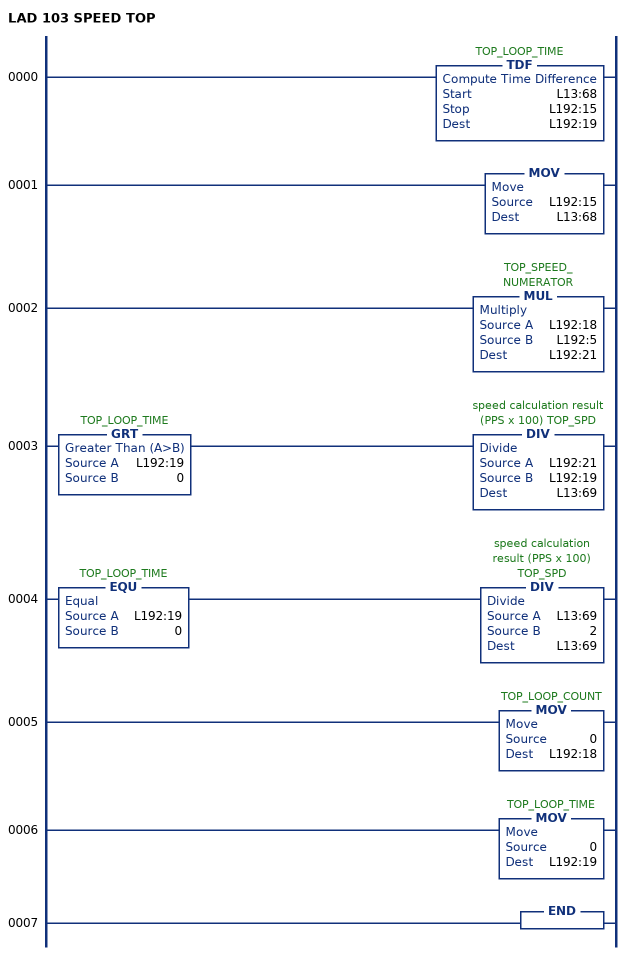
% Rung: 0 %
SOR TDF L13:68 L192:15 L192:19 EOR
%   L192:15  TOP_THIS_TIME  "rtc top belt movement event time" %
%   L192:19  TOP_LOOP_TIME %
% Rung: 1 %
SOR MOV L192:15 L13:68 EOR
%   L192:15  TOP_THIS_TIME  "rtc top belt movement event time" %
% Rung: 2 %
SOR MUL L192:18 L192:5 L192:21 EOR
%   L192:18  TOP_LOOP_COUNT %
%   L192:5  TKS_PER_SECOND %
%   L192:21  TOP_SPEED_NUMERATOR %
% Rung: 3 %
SOR GRT L192:19 0 DIV L192:21 L192:19 L13:69 EOR
%   L192:19  TOP_LOOP_TIME %
%   L192:21  TOP_SPEED_NUMERATOR %
%   L13:69  TOP_SPD  "speed calculation result (PPS x 100)" %
% Rung: 4 %
SOR EQU L192:19 0 DIV L13:69 2 L13:69 EOR
%   L192:19  TOP_LOOP_TIME %
%   L13:69  TOP_SPD  "speed calculation result (PPS x 100)" %
% Rung: 5 %
SOR MOV 0 L192:18 EOR
%   L192:18  TOP_LOOP_COUNT %
% Rung: 6 %
SOR MOV 0 L192:19 EOR
%   L192:19  TOP_LOOP_TIME %
% Rung: 7 %
SOR END EOR

LADDER 105 "P TOP"    % high speed %
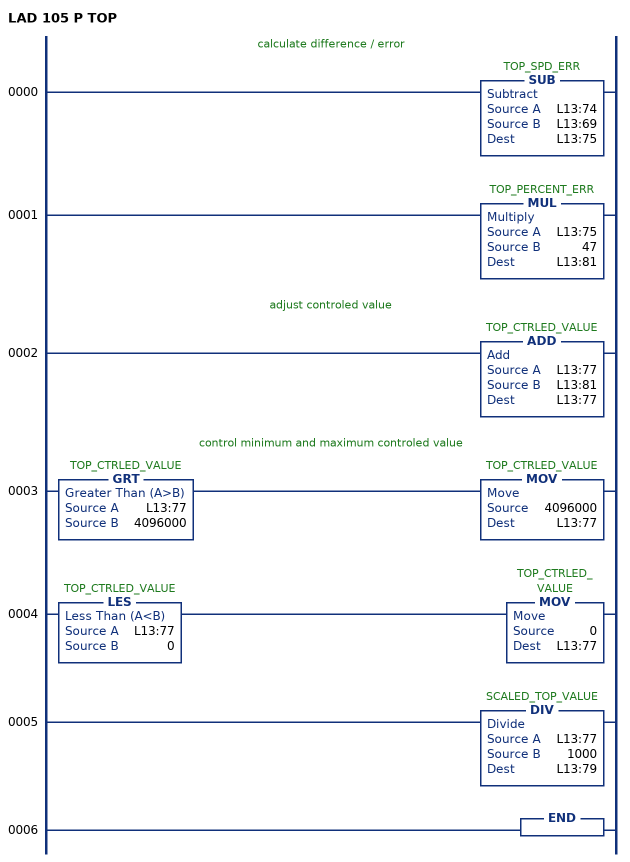
% Rung: 0 %
% calculate difference / error %
SOR SUB L13:74 L13:69 L13:75 EOR
%   L13:74  TOP_SPD_SETPOINT %
%   L13:69  TOP_SPD  "speed calculation result (PPS x 100)" %
%   L13:75  TOP_SPD_ERR %
% Rung: 1 %
SOR MUL L13:75 47 L13:81 EOR
%   L13:75  TOP_SPD_ERR %
%   L13:81  TOP_PERCENT_ERR %
% Rung: 2 %
% adjust controled value %
SOR ADD L13:77 L13:81 L13:77 EOR
%   L13:77  TOP_CTRLED_VALUE %
%   L13:81  TOP_PERCENT_ERR %
% Rung: 3 %
% control minimum and maximum controled value %
SOR GRT L13:77 4096000 MOV 4096000 L13:77 EOR
%   L13:77  TOP_CTRLED_VALUE %
% Rung: 4 %
SOR LES L13:77 0 MOV 0 L13:77 EOR
%   L13:77  TOP_CTRLED_VALUE %
% Rung: 5 %
SOR DIV L13:77 1000 L13:79 EOR
%   L13:77  TOP_CTRLED_VALUE %
%   L13:79  SCALED_TOP_VALUE %
% Rung: 6 %
SOR END EOR

LADDER 111 "SHIFT TOP"
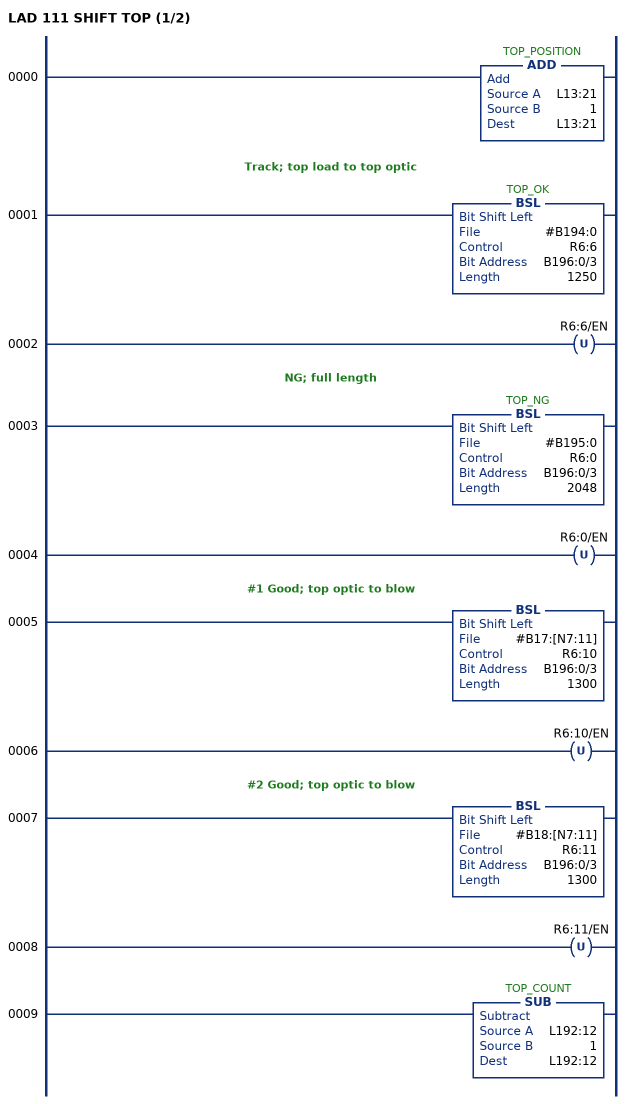
% Rung: 0 %
SOR ADD L13:21 1 L13:21 EOR
%   L13:21  TOP_POSITION %
% Rung: 1 %
% TITLE: Track; top load to top optic %
SOR BSL #B194:0 R6:6 B196:0/3 1250 EOR
%   B194:0  TOP_OK %
%   B196:0/3  OFF %
% Rung: 2 %
SOR OTU R6:6/EN EOR
% Rung: 3 %
% TITLE: NG; full length %
SOR BSL #B195:0 R6:0 B196:0/3 2048 EOR
%   B195:0  TOP_NG %
%   B196:0/3  OFF %
% Rung: 4 %
SOR OTU R6:0/EN EOR
% Rung: 5 %
% TITLE: #1 Good; top optic to blow %
SOR BSL #B17:[N7:11] R6:10 B196:0/3 1300 EOR
%   B196:0/3  OFF %
% Rung: 6 %
SOR OTU R6:10/EN EOR
% Rung: 7 %
% TITLE: #2 Good; top optic to blow %
SOR BSL #B18:[N7:11] R6:11 B196:0/3 1300 EOR
%   B196:0/3  OFF %
% Rung: 8 %
SOR OTU R6:11/EN EOR
% Rung: 9 %
SOR SUB L192:12 1 L192:12 EOR
%   L192:12  TOP_COUNT %

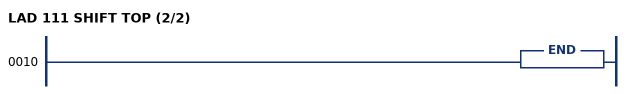
% Rung: 10 %
SOR END EOR

LADDER 131 "READXFER"
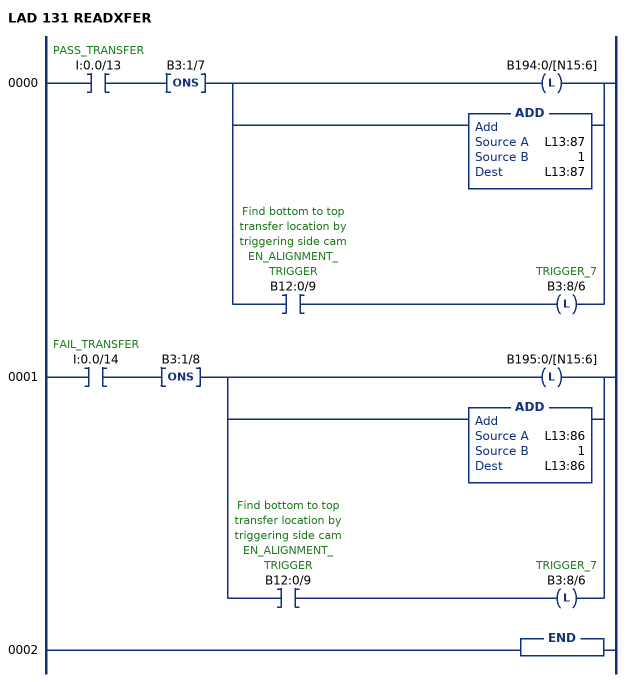
% Rung: 0 %
SOR XIC I:0.0/13 ONS B3:1/7 BST OTL B194:0/[N15:6] NXB ADD L13:87 1 L13:87 NXB XIC B12:0/9 OTL B3:8/6 BND EOR
%   I:0.0/13  PASS_TRANSFER %
%   B194:0  TOP_OK %
%   N15:6  XFER_IN_LOC %
%   B12:0/9  EN_ALIGNMENT_TRIGGER  "Find bottom to top transfer location by triggering side cam" %
%   B3:8/6  TRIGGER_7 %
% Rung: 1 %
SOR XIC I:0.0/14 ONS B3:1/8 BST OTL B195:0/[N15:6] NXB ADD L13:86 1 L13:86 NXB XIC B12:0/9 OTL B3:8/6 BND EOR
%   I:0.0/14  FAIL_TRANSFER %
%   B195:0  TOP_NG %
%   N15:6  XFER_IN_LOC %
%   B12:0/9  EN_ALIGNMENT_TRIGGER  "Find bottom to top transfer location by triggering side cam" %
%   B3:8/6  TRIGGER_7 %
% Rung: 2 %
SOR END EOR

LADDER 138 "BYPASTOPOP"
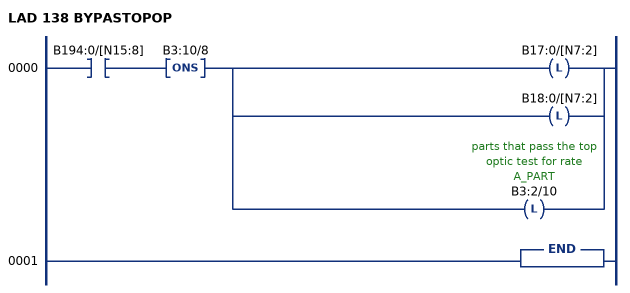
% Rung: 0 %
SOR XIC B194:0/[N15:8] ONS B3:10/8 BST OTL B17:0/[N7:2] NXB OTL B18:0/[N7:2] NXB OTL B3:2/10 BND EOR
%   B194:0  TOP_OK %
%   N15:8  TOP_OPTIC_LOC %
%   B17:0  GOOD1 %
%   N7:2  TOP_OPT_LOAD_LOC  "part load location" %
%   B18:0  GOOD2 %
%   B3:2/10  A_PART  "parts that pass the top optic test for rate" %
% Rung: 1 %
SOR END EOR

LADDER 140 "TOP_OPTIC"
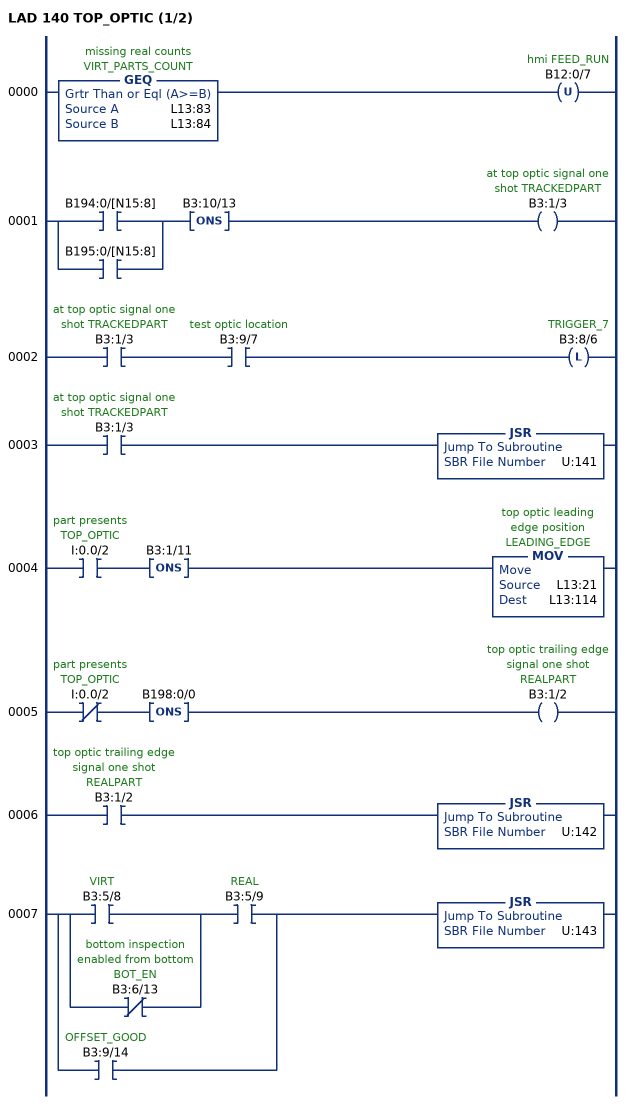
% Rung: 0 %
SOR GEQ L13:83 L13:84 OTU B12:0/7 EOR
%   L13:83  VIRT_PARTS_COUNT  "missing real counts" %
%   L13:84  FELL_PARTS_LIMIT %
%   B12:0/7  FEED_RUN  "hmi" %
% Rung: 1 %
SOR BST XIC B194:0/[N15:8] NXB XIC B195:0/[N15:8] BND ONS B3:10/13 OTE B3:1/3 EOR
%   B194:0  TOP_OK %
%   N15:8  TOP_OPTIC_LOC %
%   B195:0  TOP_NG %
%   B3:1/3  TRACKEDPART  "at top optic signal one shot" %
% Rung: 2 %
SOR XIC B3:1/3 XIC B3:9/7 OTL B3:8/6 EOR
%   B3:1/3  TRACKEDPART  "at top optic signal one shot" %
%   B3:9/7  "test optic location" %
%   B3:8/6  TRIGGER_7 %
% Rung: 3 %
SOR XIC B3:1/3 JSR U:141 EOR
%   B3:1/3  TRACKEDPART  "at top optic signal one shot" %
% Rung: 4 %
SOR XIC I:0.0/2 ONS B3:1/11 MOV L13:21 L13:114 EOR
%   I:0.0/2  TOP_OPTIC  "part presents" %
%   L13:21  TOP_POSITION %
%   L13:114  LEADING_EDGE  "top optic leading edge position" %
% Rung: 5 %
SOR XIO I:0.0/2 ONS B198:0/0 OTE B3:1/2 EOR
%   I:0.0/2  TOP_OPTIC  "part presents" %
%   B3:1/2  REALPART  "top optic trailing edge signal one shot" %
% Rung: 6 %
SOR XIC B3:1/2 JSR U:142 EOR
%   B3:1/2  REALPART  "top optic trailing edge signal one shot" %
% Rung: 7 %
SOR BST BST XIC B3:5/8 NXB XIO B3:6/13 BND XIC B3:5/9 NXB XIC B3:9/14 BND JSR U:143 EOR
%   B3:5/8  VIRT %
%   B3:6/13  BOT_EN  "bottom inspection enabled from bottom" %
%   B3:5/9  REAL %
%   B3:9/14  OFFSET_GOOD %

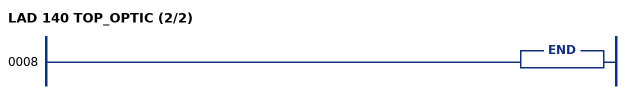
% Rung: 8 %
SOR END EOR

LADDER 141 "TOPOP_VERT"
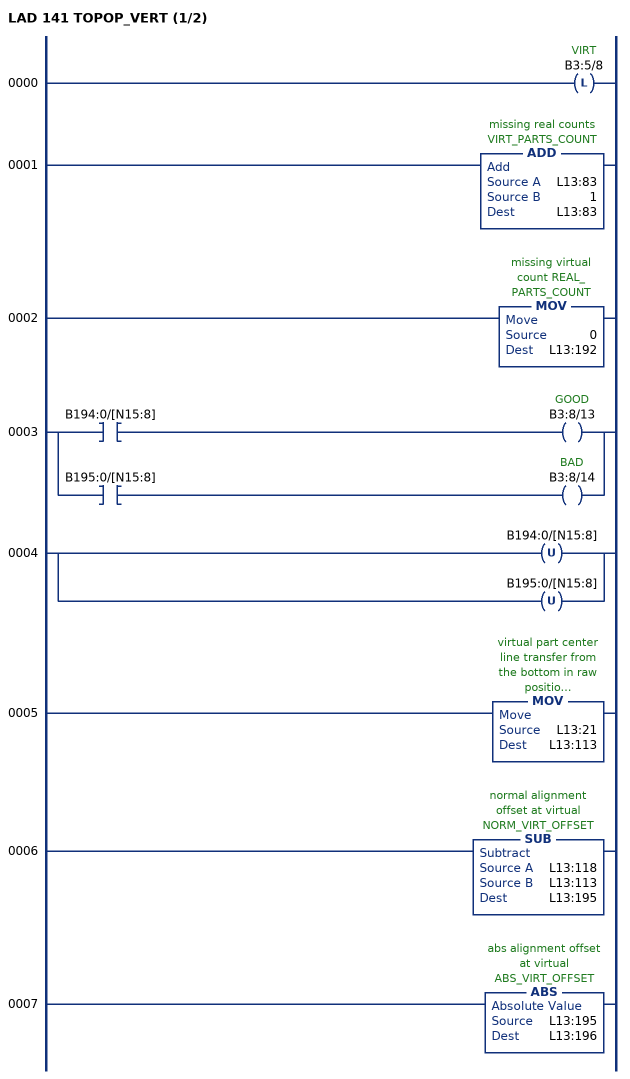
% Rung: 0 %
SOR OTL B3:5/8 EOR
%   B3:5/8  VIRT %
% Rung: 1 %
SOR ADD L13:83 1 L13:83 EOR
%   L13:83  VIRT_PARTS_COUNT  "missing real counts" %
% Rung: 2 %
SOR MOV 0 L13:192 EOR
%   L13:192  REAL_PARTS_COUNT  "missing virtual count" %
% Rung: 3 %
SOR BST XIC B194:0/[N15:8] OTE B3:8/13 NXB XIC B195:0/[N15:8] OTE B3:8/14 BND EOR
%   B194:0  TOP_OK %
%   N15:8  TOP_OPTIC_LOC %
%   B3:8/13  GOOD %
%   B195:0  TOP_NG %
%   B3:8/14  BAD %
% Rung: 4 %
SOR BST OTU B194:0/[N15:8] NXB OTU B195:0/[N15:8] BND EOR
%   B194:0  TOP_OK %
%   N15:8  TOP_OPTIC_LOC %
%   B195:0  TOP_NG %
% Rung: 5 %
SOR MOV L13:21 L13:113 EOR
%   L13:21  TOP_POSITION %
%   L13:113  VERTUAL_CL_POSITION  "virtual part center line transfer from the bottom in raw position" %
% Rung: 6 %
SOR SUB L13:118 L13:113 L13:195 EOR
%   L13:118  REAL_CL_POSITION  "real part center line in raw position" %
%   L13:113  VERTUAL_CL_POSITION  "virtual part center line transfer from the bottom in raw position" %
%   L13:195  NORM_VIRT_OFFSET  "normal alignment offset at virtual" %
% Rung: 7 %
SOR ABS L13:195 L13:196 EOR
%   L13:195  NORM_VIRT_OFFSET  "normal alignment offset at virtual" %
%   L13:196  ABS_VIRT_OFFSET  "abs alignment offset at virtual" %

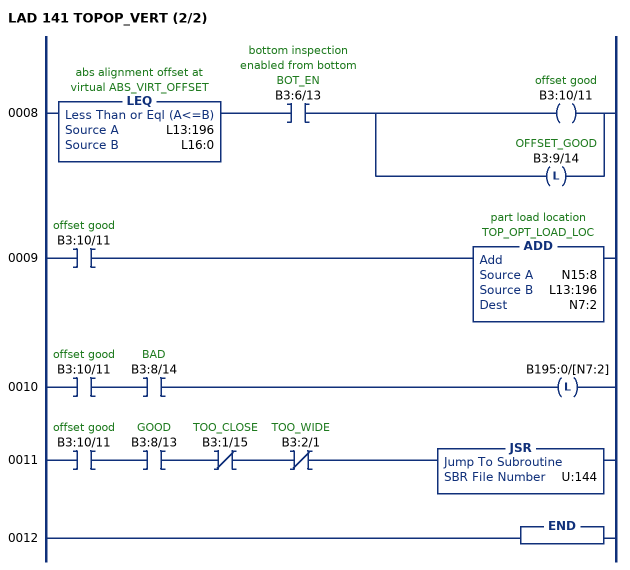
% Rung: 8 %
SOR LEQ L13:196 L16:0 XIC B3:6/13 BST OTE B3:10/11 NXB OTL B3:9/14 BND EOR
%   L13:196  ABS_VIRT_OFFSET  "abs alignment offset at virtual" %
%   L16:0  MAX_OFFSET %
%   B3:6/13  BOT_EN  "bottom inspection enabled from bottom" %
%   B3:10/11  "offset good" %
%   B3:9/14  OFFSET_GOOD %
% Rung: 9 %
SOR XIC B3:10/11 ADD N15:8 L13:196 N7:2 EOR
%   B3:10/11  "offset good" %
%   N15:8  TOP_OPTIC_LOC %
%   L13:196  ABS_VIRT_OFFSET  "abs alignment offset at virtual" %
%   N7:2  TOP_OPT_LOAD_LOC  "part load location" %
% Rung: 10 %
SOR XIC B3:10/11 XIC B3:8/14 OTL B195:0/[N7:2] EOR
%   B3:10/11  "offset good" %
%   B3:8/14  BAD %
%   B195:0  TOP_NG %
%   N7:2  TOP_OPT_LOAD_LOC  "part load location" %
% Rung: 11 %
SOR XIC B3:10/11 XIC B3:8/13 XIO B3:1/15 XIO B3:2/1 JSR U:144 EOR
%   B3:10/11  "offset good" %
%   B3:8/13  GOOD %
%   B3:1/15  TOO_CLOSE %
%   B3:2/1  TOO_WIDE %
% Rung: 12 %
SOR END EOR

LADDER 142 "TOPOP_REAL"
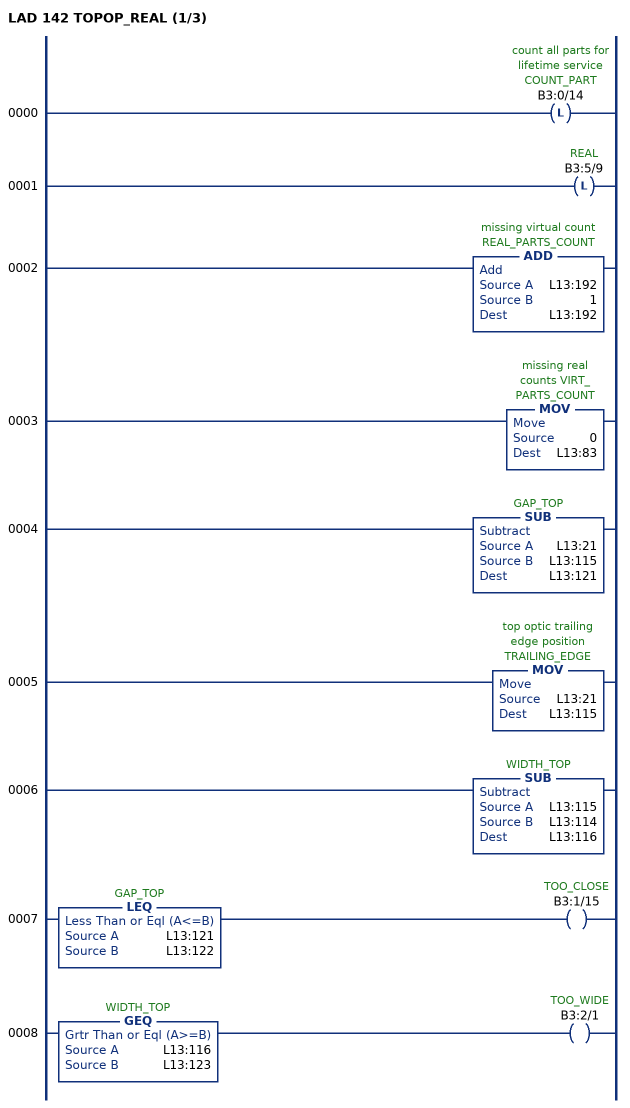
% Rung: 0 %
SOR OTL B3:0/14 EOR
%   B3:0/14  COUNT_PART  "count all parts for lifetime service" %
% Rung: 1 %
SOR OTL B3:5/9 EOR
%   B3:5/9  REAL %
% Rung: 2 %
SOR ADD L13:192 1 L13:192 EOR
%   L13:192  REAL_PARTS_COUNT  "missing virtual count" %
% Rung: 3 %
SOR MOV 0 L13:83 EOR
%   L13:83  VIRT_PARTS_COUNT  "missing real counts" %
% Rung: 4 %
SOR SUB L13:21 L13:115 L13:121 EOR
%   L13:21  TOP_POSITION %
%   L13:115  TRAILING_EDGE  "top optic trailing edge position" %
%   L13:121  GAP_TOP %
% Rung: 5 %
SOR MOV L13:21 L13:115 EOR
%   L13:21  TOP_POSITION %
%   L13:115  TRAILING_EDGE  "top optic trailing edge position" %
% Rung: 6 %
SOR SUB L13:115 L13:114 L13:116 EOR
%   L13:115  TRAILING_EDGE  "top optic trailing edge position" %
%   L13:114  LEADING_EDGE  "top optic leading edge position" %
%   L13:116  WIDTH_TOP %
% Rung: 7 %
SOR LEQ L13:121 L13:122 OTE B3:1/15 EOR
%   L13:121  GAP_TOP %
%   L13:122  TOP_MIN_GAP %
%   B3:1/15  TOO_CLOSE %
% Rung: 8 %
SOR GEQ L13:116 L13:123 OTE B3:2/1 EOR
%   L13:116  WIDTH_TOP %
%   L13:123  TOP_MAX_WIDTH %
%   B3:2/1  TOO_WIDE %

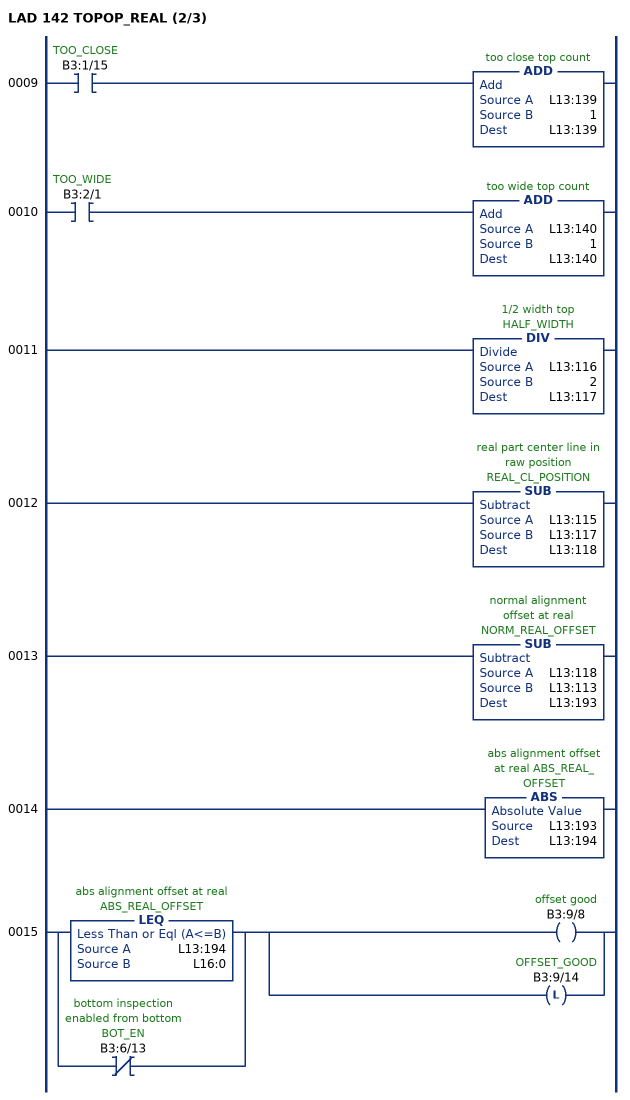
% Rung: 9 %
SOR XIC B3:1/15 ADD L13:139 1 L13:139 EOR
%   B3:1/15  TOO_CLOSE %
%   L13:139  "too close top count" %
% Rung: 10 %
SOR XIC B3:2/1 ADD L13:140 1 L13:140 EOR
%   B3:2/1  TOO_WIDE %
%   L13:140  "too wide top count" %
% Rung: 11 %
SOR DIV L13:116 2 L13:117 EOR
%   L13:116  WIDTH_TOP %
%   L13:117  HALF_WIDTH  "1/2 width top" %
% Rung: 12 %
SOR SUB L13:115 L13:117 L13:118 EOR
%   L13:115  TRAILING_EDGE  "top optic trailing edge position" %
%   L13:117  HALF_WIDTH  "1/2 width top" %
%   L13:118  REAL_CL_POSITION  "real part center line in raw position" %
% Rung: 13 %
SOR SUB L13:118 L13:113 L13:193 EOR
%   L13:118  REAL_CL_POSITION  "real part center line in raw position" %
%   L13:113  VERTUAL_CL_POSITION  "virtual part center line transfer from the bottom in raw position" %
%   L13:193  NORM_REAL_OFFSET  "normal alignment offset at real" %
% Rung: 14 %
SOR ABS L13:193 L13:194 EOR
%   L13:193  NORM_REAL_OFFSET  "normal alignment offset at real" %
%   L13:194  ABS_REAL_OFFSET  "abs alignment offset at real" %
% Rung: 15 %
SOR BST LEQ L13:194 L16:0 NXB XIO B3:6/13 BND BST OTE B3:9/8 NXB OTL B3:9/14 BND EOR
%   L13:194  ABS_REAL_OFFSET  "abs alignment offset at real" %
%   L16:0  MAX_OFFSET %
%   B3:6/13  BOT_EN  "bottom inspection enabled from bottom" %
%   B3:9/8  "offset good" %
%   B3:9/14  OFFSET_GOOD %

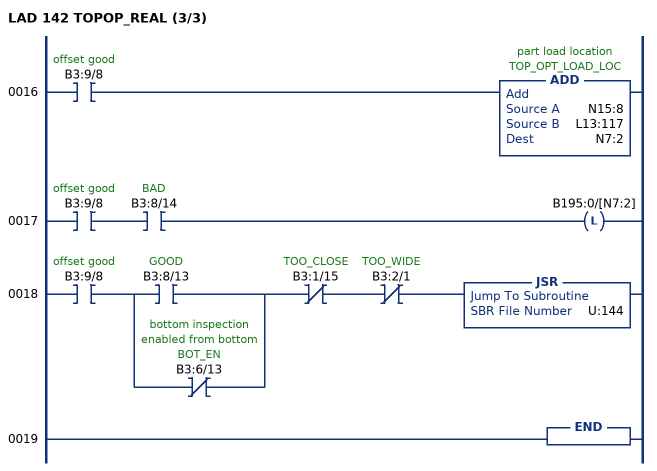
% Rung: 16 %
SOR XIC B3:9/8 ADD N15:8 L13:117 N7:2 EOR
%   B3:9/8  "offset good" %
%   N15:8  TOP_OPTIC_LOC %
%   L13:117  HALF_WIDTH  "1/2 width top" %
%   N7:2  TOP_OPT_LOAD_LOC  "part load location" %
% Rung: 17 %
SOR XIC B3:9/8 XIC B3:8/14 OTL B195:0/[N7:2] EOR
%   B3:9/8  "offset good" %
%   B3:8/14  BAD %
%   B195:0  TOP_NG %
%   N7:2  TOP_OPT_LOAD_LOC  "part load location" %
% Rung: 18 %
SOR XIC B3:9/8 BST XIC B3:8/13 NXB XIO B3:6/13 BND XIO B3:1/15 XIO B3:2/1 JSR U:144 EOR
%   B3:9/8  "offset good" %
%   B3:8/13  GOOD %
%   B3:6/13  BOT_EN  "bottom inspection enabled from bottom" %
%   B3:1/15  TOO_CLOSE %
%   B3:2/1  TOO_WIDE %
% Rung: 19 %
SOR END EOR

LADDER 143 "CT ALIGNS"
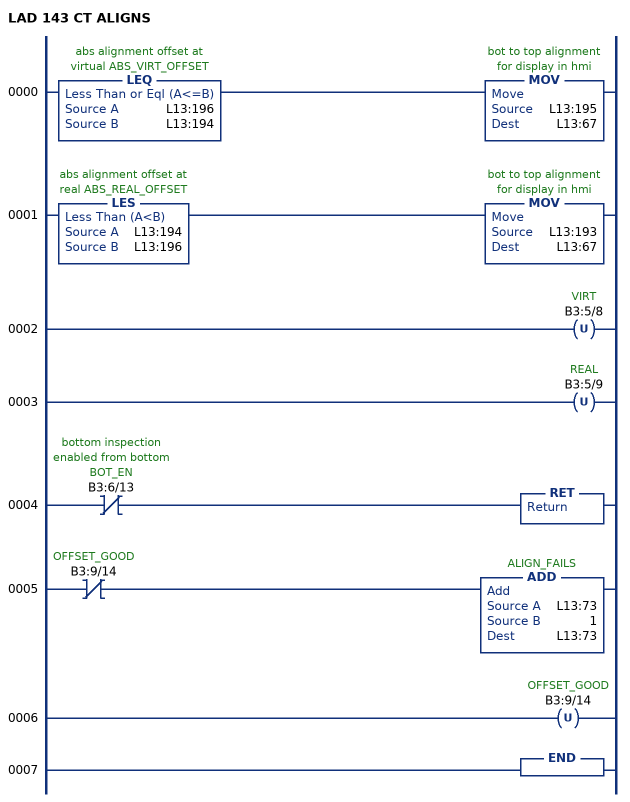
% Rung: 0 %
SOR LEQ L13:196 L13:194 MOV L13:195 L13:67 EOR
%   L13:196  ABS_VIRT_OFFSET  "abs alignment offset at virtual" %
%   L13:194  ABS_REAL_OFFSET  "abs alignment offset at real" %
%   L13:195  NORM_VIRT_OFFSET  "normal alignment offset at virtual" %
%   L13:67  "bot to top alignment for display in hmi" %
% Rung: 1 %
SOR LES L13:194 L13:196 MOV L13:193 L13:67 EOR
%   L13:194  ABS_REAL_OFFSET  "abs alignment offset at real" %
%   L13:196  ABS_VIRT_OFFSET  "abs alignment offset at virtual" %
%   L13:193  NORM_REAL_OFFSET  "normal alignment offset at real" %
%   L13:67  "bot to top alignment for display in hmi" %
% Rung: 2 %
SOR OTU B3:5/8 EOR
%   B3:5/8  VIRT %
% Rung: 3 %
SOR OTU B3:5/9 EOR
%   B3:5/9  REAL %
% Rung: 4 %
SOR XIO B3:6/13 RET EOR
%   B3:6/13  BOT_EN  "bottom inspection enabled from bottom" %
% Rung: 5 %
SOR XIO B3:9/14 ADD L13:73 1 L13:73 EOR
%   B3:9/14  OFFSET_GOOD %
%   L13:73  ALIGN_FAILS %
% Rung: 6 %
SOR OTU B3:9/14 EOR
%   B3:9/14  OFFSET_GOOD %
% Rung: 7 %
SOR END EOR

LADDER 144 "SET GOOD"
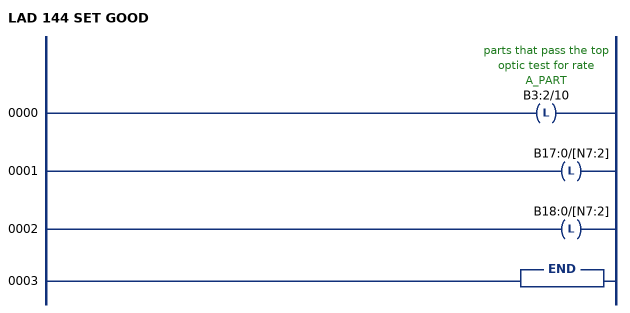
% Rung: 0 %
SOR OTL B3:2/10 EOR
%   B3:2/10  A_PART  "parts that pass the top optic test for rate" %
% Rung: 1 %
SOR OTL B17:0/[N7:2] EOR
%   B17:0  GOOD1 %
%   N7:2  TOP_OPT_LOAD_LOC  "part load location" %
% Rung: 2 %
SOR OTL B18:0/[N7:2] EOR
%   B18:0  GOOD2 %
%   N7:2  TOP_OPT_LOAD_LOC  "part load location" %
% Rung: 3 %
SOR END EOR

LADDER 150 "TOP_OPTIC"
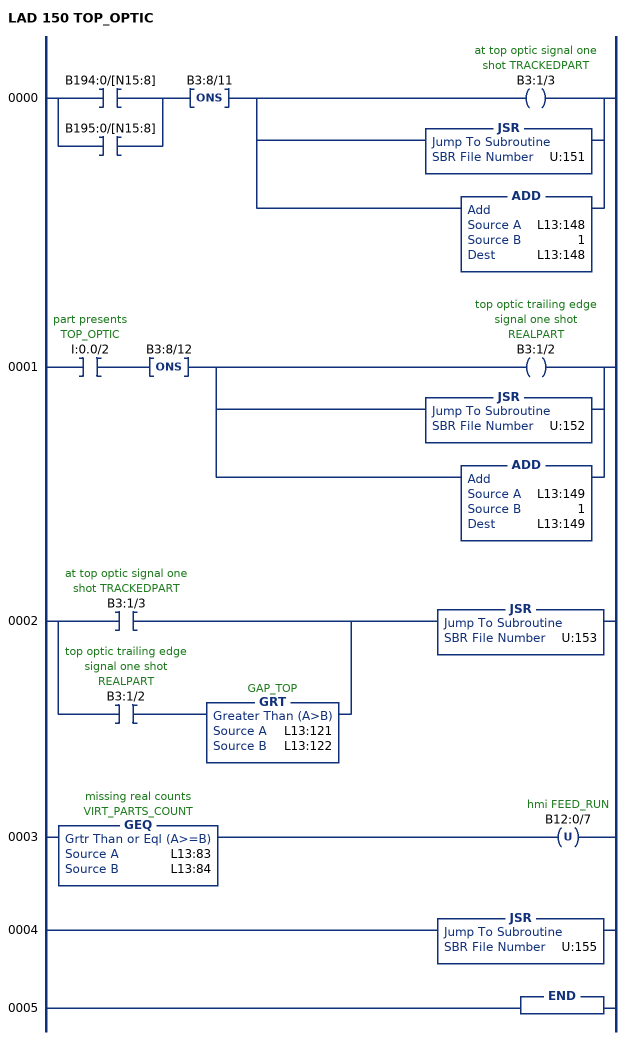
% Rung: 0 %
SOR BST XIC B194:0/[N15:8] NXB XIC B195:0/[N15:8] BND ONS B3:8/11 BST OTE B3:1/3 NXB JSR U:151 NXB ADD L13:148 1 L13:148 BND EOR
%   B194:0  TOP_OK %
%   N15:8  TOP_OPTIC_LOC %
%   B195:0  TOP_NG %
%   B3:1/3  TRACKEDPART  "at top optic signal one shot" %
% Rung: 1 %
SOR XIC I:0.0/2 ONS B3:8/12 BST OTE B3:1/2 NXB JSR U:152 NXB ADD L13:149 1 L13:149 BND EOR
%   I:0.0/2  TOP_OPTIC  "part presents" %
%   B3:1/2  REALPART  "top optic trailing edge signal one shot" %
% Rung: 2 %
SOR BST XIC B3:1/3 NXB XIC B3:1/2 GRT L13:121 L13:122 BND JSR U:153 EOR
%   B3:1/3  TRACKEDPART  "at top optic signal one shot" %
%   B3:1/2  REALPART  "top optic trailing edge signal one shot" %
%   L13:121  GAP_TOP %
%   L13:122  TOP_MIN_GAP %
% Rung: 3 %
SOR GEQ L13:83 L13:84 OTU B12:0/7 EOR
%   L13:83  VIRT_PARTS_COUNT  "missing real counts" %
%   L13:84  FELL_PARTS_LIMIT %
%   B12:0/7  FEED_RUN  "hmi" %
% Rung: 4 %
SOR JSR U:155 EOR
% Rung: 5 %
SOR END EOR

LADDER 151 "TOPOP_VERT"
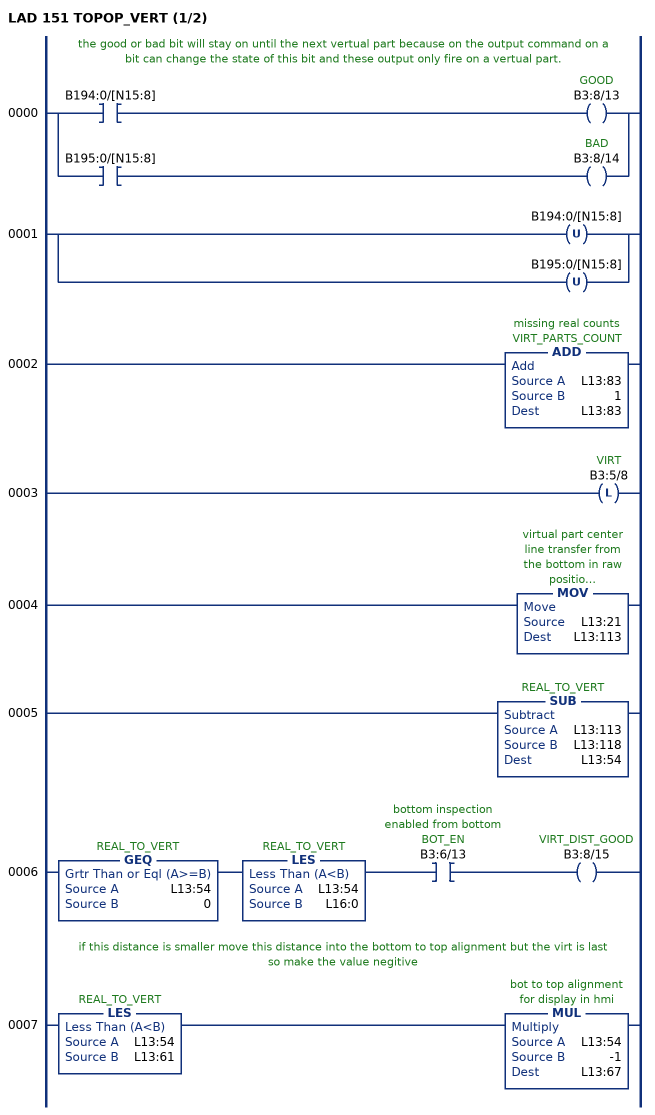
% Rung: 0 %
% the good or bad bit will stay on until the next vertual part because on the output command on a bit can change the state of this bit and these output only fire on a vertual part. %
SOR BST XIC B194:0/[N15:8] OTE B3:8/13 NXB XIC B195:0/[N15:8] OTE B3:8/14 BND EOR
%   B194:0  TOP_OK %
%   N15:8  TOP_OPTIC_LOC %
%   B3:8/13  GOOD %
%   B195:0  TOP_NG %
%   B3:8/14  BAD %
% Rung: 1 %
SOR BST OTU B194:0/[N15:8] NXB OTU B195:0/[N15:8] BND EOR
%   B194:0  TOP_OK %
%   N15:8  TOP_OPTIC_LOC %
%   B195:0  TOP_NG %
% Rung: 2 %
SOR ADD L13:83 1 L13:83 EOR
%   L13:83  VIRT_PARTS_COUNT  "missing real counts" %
% Rung: 3 %
SOR OTL B3:5/8 EOR
%   B3:5/8  VIRT %
% Rung: 4 %
SOR MOV L13:21 L13:113 EOR
%   L13:21  TOP_POSITION %
%   L13:113  VERTUAL_CL_POSITION  "virtual part center line transfer from the bottom in raw position" %
% Rung: 5 %
SOR SUB L13:113 L13:118 L13:54 EOR
%   L13:113  VERTUAL_CL_POSITION  "virtual part center line transfer from the bottom in raw position" %
%   L13:118  REAL_CL_POSITION  "real part center line in raw position" %
%   L13:54  REAL_TO_VERT %
% Rung: 6 %
SOR GEQ L13:54 0 LES L13:54 L16:0 XIC B3:6/13 OTE B3:8/15 EOR
%   L13:54  REAL_TO_VERT %
%   L16:0  MAX_OFFSET %
%   B3:6/13  BOT_EN  "bottom inspection enabled from bottom" %
%   B3:8/15  VIRT_DIST_GOOD %
% Rung: 7 %
% if this distance is smaller move this distance into the bottom to top alignment but the virt is last so make the value negitive %
SOR LES L13:54 L13:61 MUL L13:54 -1 L13:67 EOR
%   L13:54  REAL_TO_VERT %
%   L13:61  VIRT_TO_REAL %
%   L13:67  "bot to top alignment for display in hmi" %

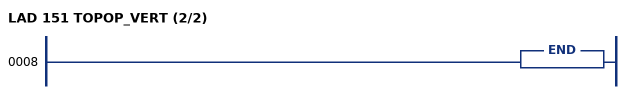
% Rung: 8 %
SOR END EOR

LADDER 152 "TOPOP_REAL"
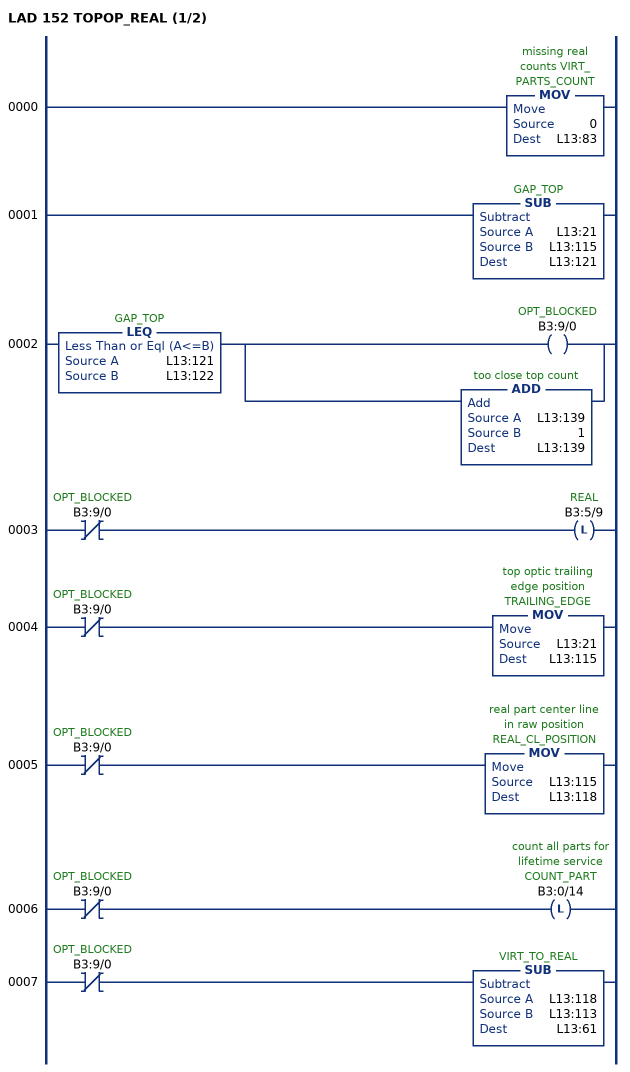
% Rung: 0 %
SOR MOV 0 L13:83 EOR
%   L13:83  VIRT_PARTS_COUNT  "missing real counts" %
% Rung: 1 %
SOR SUB L13:21 L13:115 L13:121 EOR
%   L13:21  TOP_POSITION %
%   L13:115  TRAILING_EDGE  "top optic trailing edge position" %
%   L13:121  GAP_TOP %
% Rung: 2 %
SOR LEQ L13:121 L13:122 BST OTE B3:9/0 NXB ADD L13:139 1 L13:139 BND EOR
%   L13:121  GAP_TOP %
%   L13:122  TOP_MIN_GAP %
%   B3:9/0  OPT_BLOCKED %
%   L13:139  "too close top count" %
% Rung: 3 %
SOR XIO B3:9/0 OTL B3:5/9 EOR
%   B3:9/0  OPT_BLOCKED %
%   B3:5/9  REAL %
% Rung: 4 %
SOR XIO B3:9/0 MOV L13:21 L13:115 EOR
%   B3:9/0  OPT_BLOCKED %
%   L13:21  TOP_POSITION %
%   L13:115  TRAILING_EDGE  "top optic trailing edge position" %
% Rung: 5 %
SOR XIO B3:9/0 MOV L13:115 L13:118 EOR
%   B3:9/0  OPT_BLOCKED %
%   L13:115  TRAILING_EDGE  "top optic trailing edge position" %
%   L13:118  REAL_CL_POSITION  "real part center line in raw position" %
% Rung: 6 %
SOR XIO B3:9/0 OTL B3:0/14 EOR
%   B3:9/0  OPT_BLOCKED %
%   B3:0/14  COUNT_PART  "count all parts for lifetime service" %
% Rung: 7 %
SOR XIO B3:9/0 SUB L13:118 L13:113 L13:61 EOR
%   B3:9/0  OPT_BLOCKED %
%   L13:118  REAL_CL_POSITION  "real part center line in raw position" %
%   L13:113  VERTUAL_CL_POSITION  "virtual part center line transfer from the bottom in raw position" %
%   L13:61  VIRT_TO_REAL %

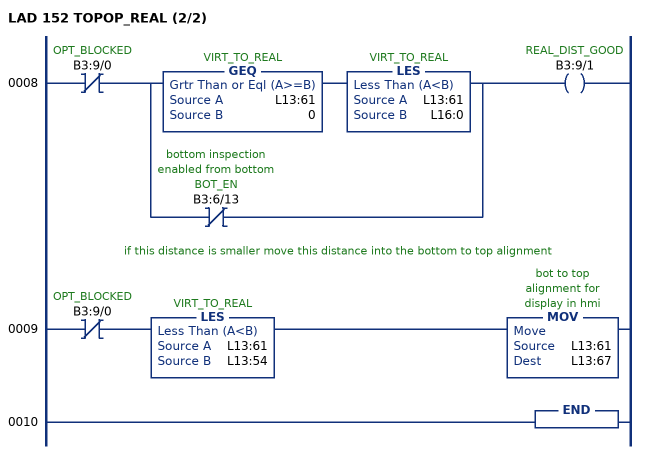
% Rung: 8 %
SOR XIO B3:9/0 BST GEQ L13:61 0 LES L13:61 L16:0 NXB XIO B3:6/13 BND OTE B3:9/1 EOR
%   B3:9/0  OPT_BLOCKED %
%   L13:61  VIRT_TO_REAL %
%   L16:0  MAX_OFFSET %
%   B3:6/13  BOT_EN  "bottom inspection enabled from bottom" %
%   B3:9/1  REAL_DIST_GOOD %
% Rung: 9 %
% if this distance is smaller move this distance into the bottom to top alignment %
SOR XIO B3:9/0 LES L13:61 L13:54 MOV L13:61 L13:67 EOR
%   B3:9/0  OPT_BLOCKED %
%   L13:61  VIRT_TO_REAL %
%   L13:54  REAL_TO_VERT %
%   L13:67  "bot to top alignment for display in hmi" %
% Rung: 10 %
SOR END EOR

LADDER 153 "TOPOP_TEST"
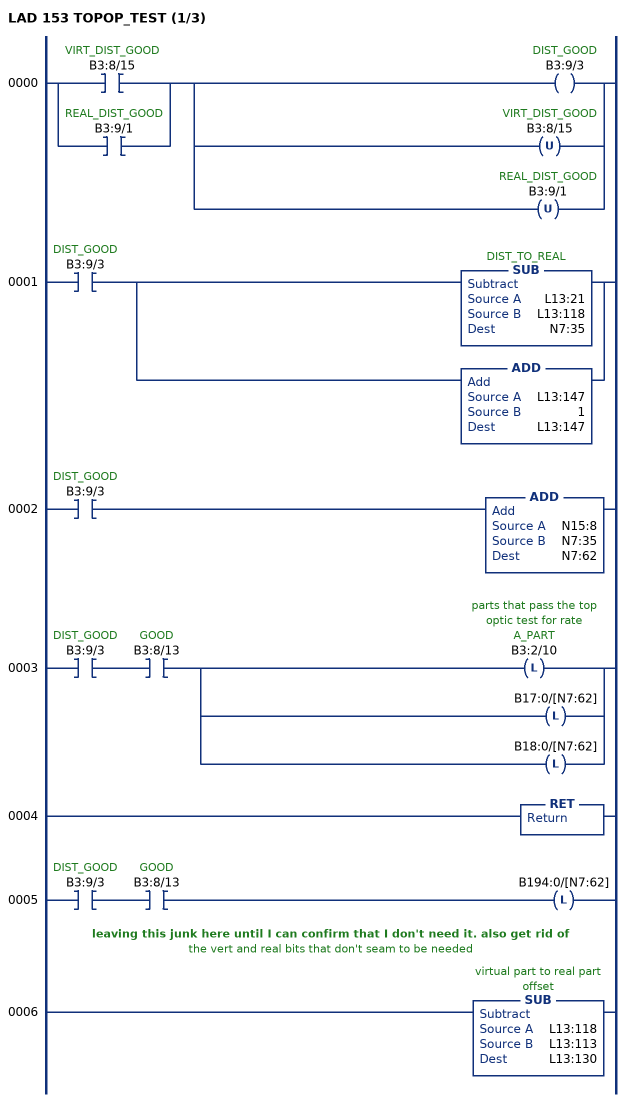
% Rung: 0 %
SOR BST XIC B3:8/15 NXB XIC B3:9/1 BND BST OTE B3:9/3 NXB OTU B3:8/15 NXB OTU B3:9/1 BND EOR
%   B3:8/15  VIRT_DIST_GOOD %
%   B3:9/1  REAL_DIST_GOOD %
%   B3:9/3  DIST_GOOD %
% Rung: 1 %
SOR XIC B3:9/3 BST SUB L13:21 L13:118 N7:35 NXB ADD L13:147 1 L13:147 BND EOR
%   B3:9/3  DIST_GOOD %
%   L13:21  TOP_POSITION %
%   L13:118  REAL_CL_POSITION  "real part center line in raw position" %
%   N7:35  DIST_TO_REAL %
% Rung: 2 %
SOR XIC B3:9/3 ADD N15:8 N7:35 N7:62 EOR
%   B3:9/3  DIST_GOOD %
%   N15:8  TOP_OPTIC_LOC %
%   N7:35  DIST_TO_REAL %
% Rung: 3 %
SOR XIC B3:9/3 XIC B3:8/13 BST OTL B3:2/10 NXB OTL B17:0/[N7:62] NXB OTL B18:0/[N7:62] BND EOR
%   B3:9/3  DIST_GOOD %
%   B3:8/13  GOOD %
%   B3:2/10  A_PART  "parts that pass the top optic test for rate" %
%   B17:0  GOOD1 %
%   B18:0  GOOD2 %
% Rung: 4 %
SOR RET EOR
% Rung: 5 %
SOR XIC B3:9/3 XIC B3:8/13 OTL B194:0/[N7:62] EOR
%   B3:9/3  DIST_GOOD %
%   B3:8/13  GOOD %
%   B194:0  TOP_OK %
% Rung: 6 %
% TITLE: leaving this junk here until I can confirm that I don't need it. also get rid of %
% the vert and real bits that don't seam to be needed %
SOR SUB L13:118 L13:113 L13:130 EOR
%   L13:118  REAL_CL_POSITION  "real part center line in raw position" %
%   L13:113  VERTUAL_CL_POSITION  "virtual part center line transfer from the bottom in raw position" %
%   L13:130  "virtual part to real part offset" %

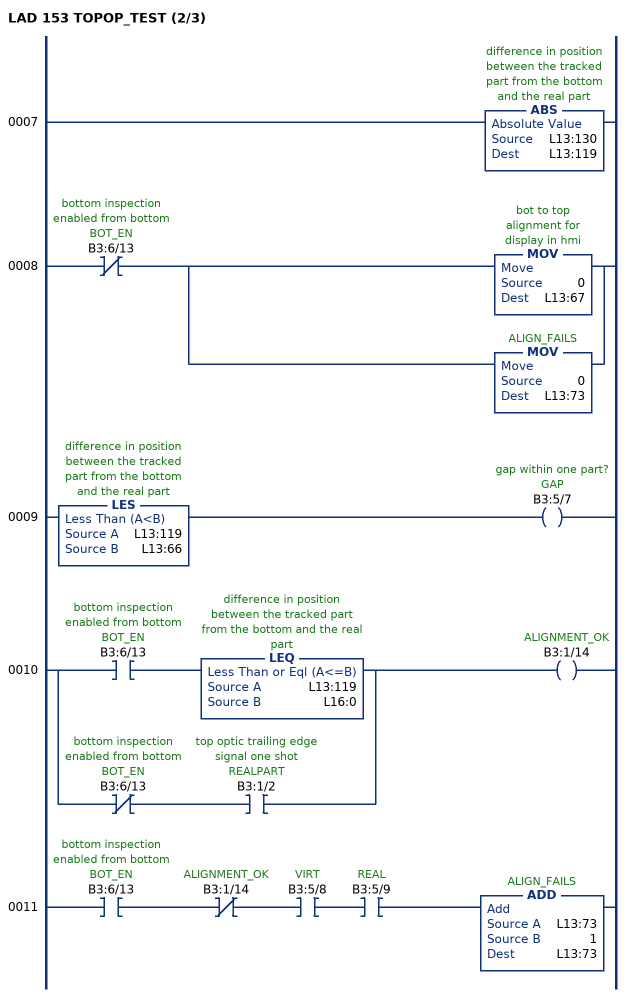
% Rung: 7 %
SOR ABS L13:130 L13:119 EOR
%   L13:130  "virtual part to real part offset" %
%   L13:119  "difference in position between the tracked part from the bottom and the real part" %
% Rung: 8 %
SOR XIO B3:6/13 BST MOV 0 L13:67 NXB MOV 0 L13:73 BND EOR
%   B3:6/13  BOT_EN  "bottom inspection enabled from bottom" %
%   L13:67  "bot to top alignment for display in hmi" %
%   L13:73  ALIGN_FAILS %
% Rung: 9 %
SOR LES L13:119 L13:66 OTE B3:5/7 EOR
%   L13:119  "difference in position between the tracked part from the bottom and the real part" %
%   L13:66  SAME_PART_GAP %
%   B3:5/7  GAP  "gap within one part?" %
% Rung: 10 %
SOR BST XIC B3:6/13 LEQ L13:119 L16:0 NXB XIO B3:6/13 XIC B3:1/2 BND OTE B3:1/14 EOR
%   B3:6/13  BOT_EN  "bottom inspection enabled from bottom" %
%   L13:119  "difference in position between the tracked part from the bottom and the real part" %
%   L16:0  MAX_OFFSET %
%   B3:1/2  REALPART  "top optic trailing edge signal one shot" %
%   B3:1/14  ALIGNMENT_OK %
% Rung: 11 %
SOR XIC B3:6/13 XIO B3:1/14 XIC B3:5/8 XIC B3:5/9 ADD L13:73 1 L13:73 EOR
%   B3:6/13  BOT_EN  "bottom inspection enabled from bottom" %
%   B3:1/14  ALIGNMENT_OK %
%   B3:5/8  VIRT %
%   B3:5/9  REAL %
%   L13:73  ALIGN_FAILS %

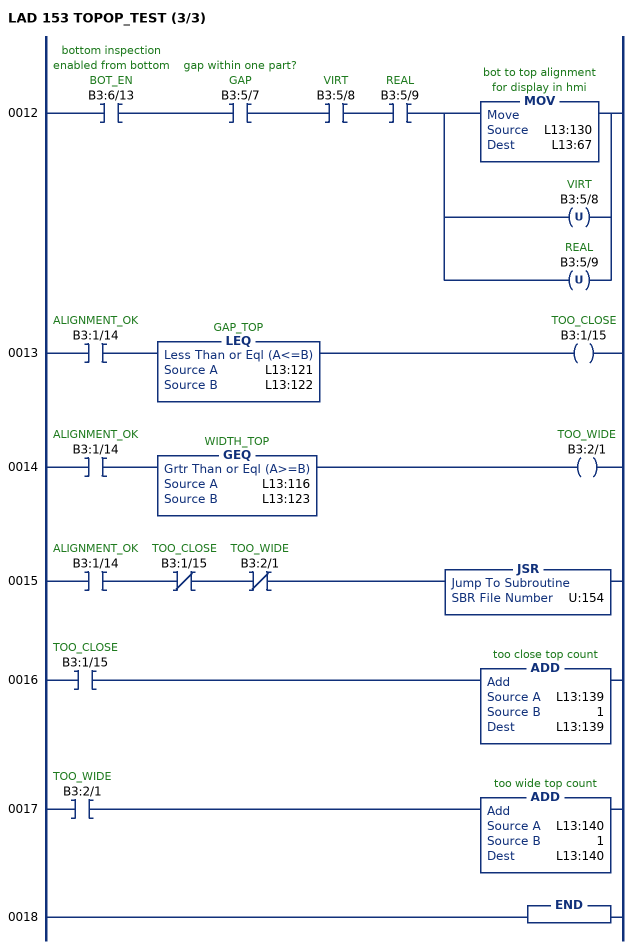
% Rung: 12 %
SOR XIC B3:6/13 XIC B3:5/7 XIC B3:5/8 XIC B3:5/9 BST MOV L13:130 L13:67 NXB OTU B3:5/8 NXB OTU B3:5/9 BND EOR
%   B3:6/13  BOT_EN  "bottom inspection enabled from bottom" %
%   B3:5/7  GAP  "gap within one part?" %
%   B3:5/8  VIRT %
%   B3:5/9  REAL %
%   L13:130  "virtual part to real part offset" %
%   L13:67  "bot to top alignment for display in hmi" %
% Rung: 13 %
SOR XIC B3:1/14 LEQ L13:121 L13:122 OTE B3:1/15 EOR
%   B3:1/14  ALIGNMENT_OK %
%   L13:121  GAP_TOP %
%   L13:122  TOP_MIN_GAP %
%   B3:1/15  TOO_CLOSE %
% Rung: 14 %
SOR XIC B3:1/14 GEQ L13:116 L13:123 OTE B3:2/1 EOR
%   B3:1/14  ALIGNMENT_OK %
%   L13:116  WIDTH_TOP %
%   L13:123  TOP_MAX_WIDTH %
%   B3:2/1  TOO_WIDE %
% Rung: 15 %
SOR XIC B3:1/14 XIO B3:1/15 XIO B3:2/1 JSR U:154 EOR
%   B3:1/14  ALIGNMENT_OK %
%   B3:1/15  TOO_CLOSE %
%   B3:2/1  TOO_WIDE %
% Rung: 16 %
SOR XIC B3:1/15 ADD L13:139 1 L13:139 EOR
%   B3:1/15  TOO_CLOSE %
%   L13:139  "too close top count" %
% Rung: 17 %
SOR XIC B3:2/1 ADD L13:140 1 L13:140 EOR
%   B3:2/1  TOO_WIDE %
%   L13:140  "too wide top count" %
% Rung: 18 %
SOR END EOR

LADDER 154 "TOP_OP_OK"
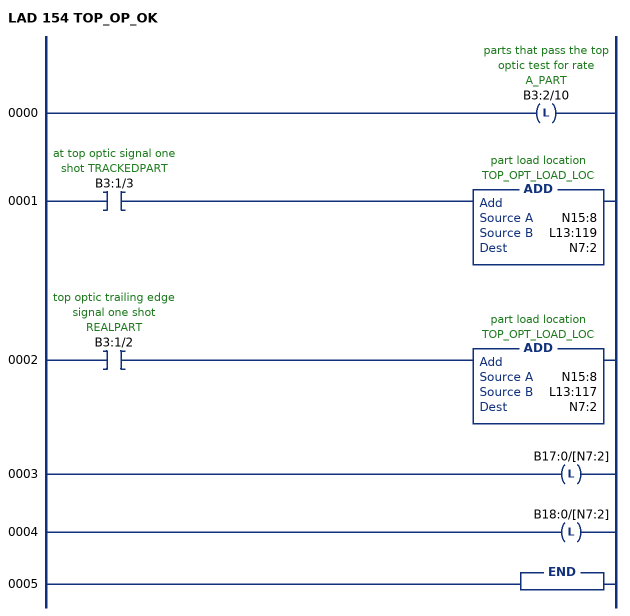
% Rung: 0 %
SOR OTL B3:2/10 EOR
%   B3:2/10  A_PART  "parts that pass the top optic test for rate" %
% Rung: 1 %
SOR XIC B3:1/3 ADD N15:8 L13:119 N7:2 EOR
%   B3:1/3  TRACKEDPART  "at top optic signal one shot" %
%   N15:8  TOP_OPTIC_LOC %
%   L13:119  "difference in position between the tracked part from the bottom and the real part" %
%   N7:2  TOP_OPT_LOAD_LOC  "part load location" %
% Rung: 2 %
SOR XIC B3:1/2 ADD N15:8 L13:117 N7:2 EOR
%   B3:1/2  REALPART  "top optic trailing edge signal one shot" %
%   N15:8  TOP_OPTIC_LOC %
%   L13:117  HALF_WIDTH  "1/2 width top" %
%   N7:2  TOP_OPT_LOAD_LOC  "part load location" %
% Rung: 3 %
SOR OTL B17:0/[N7:2] EOR
%   B17:0  GOOD1 %
%   N7:2  TOP_OPT_LOAD_LOC  "part load location" %
% Rung: 4 %
SOR OTL B18:0/[N7:2] EOR
%   B18:0  GOOD2 %
%   N7:2  TOP_OPT_LOAD_LOC  "part load location" %
% Rung: 5 %
SOR END EOR

LADDER 155 "OP RNG TST"
